FUNCTION F_LeakMonitor_LIR_2 : FB_LeakMonitor
VAR_INPUT
END_VAR
VAR_OUTPUT
	// Provide stBoundaries output so test functions can reuse the boundaries
	stBoundaries : ST_LeakBoundaries := F_LeakBoundaries();
END_VAR
VAR
	fbLeakMonitor : FB_LeakMonitor;
END_VAR

fbLeakMonitor(
	bLeakDetected := TRUE,
	nLocationResistance := stBoundaries.nLMin6,
	stBoundaries := stBoundaries
);

F_LeakMonitor_LIR_2 := fbLeakMonitor;

END_FUNCTION

(* stored: Version 1.1.0.1, ProductVersion 3.1.4020.14
   POU F_LeakMonitor_LIR_2: Id {d6bae869-88f4-4167-a80f-9e33ee99991e}, SpecialFunc None *)
